TYPE TYP_VALVE_53_HW_IN :
STRUCT
	ReachedHP AT %I* : BOOL;
	ReachedWP AT %I* : BOOL;
END_STRUCT
END_TYPE

(* stored: Version 1.1.0.1, ProductVersion 3.1.4024.12
   DUT TYP_VALVE_53_HW_IN: Id {c5e13aa1-7c5c-4628-88e3-b976d26d0ad1} *)
